Staubli VAL3: OnF1.pgx

program OnF1()
begin
  //
  if nType==1
    call setTool(sItem)
    popUpMsg("选择工具："+sItem)
  endIf

end
